Staubli VAL3: USERPAGE.pjx

--- USERPAGE.pjx ---
Parameters version=s7.6 stackSize=5000 millimeterUnit=true
Program file=changeValue.pgx
Program file=clear.pgx
Program file=divideString.pgx
Program file=editNumField.pgx
Program file=example.pgx
Program file=findPos.pgx
Program file=getListPosition.pgx
Program file=getMenu.pgx
Program file=getView.pgx
Program file=insertDialog.pgx
Program file=isListEmpty.pgx
Program file=leftPos.pgx
Program file=listadd.pgx
Program file=listcreate.pgx
Program file=listcursor.pgx
Program file=listdel.pgx
Program file=listempty.pgx
Program file=listevent.pgx
Program file=listframe.pgx
Program file=listins.pgx
Program file=listredraw.pgx
Program file=listupdate.pgx
Program file=midPos.pgx
Program file=nullKey.pgx
Program file=numCopy.pgx
Program file=printScroll.pgx
Program file=questionDialog.pgx
Program file=read.pgx
Program file=rightPos.pgx
Program file=scroll.pgx
Program file=selectNewField.pgx
Program file=setCenter.pgx
Program file=setMenu.pgx
Program file=setSizeList.pgx
Program file=setView.pgx
Program file=showBoolStatus.pgx
Program file=strfill.pgx
Program file=strfillchr.pgx
Program file=stringCopy.pgx
Program file=stringToArray.pgx
Program file=strlength.pgx
Program file=timerDialog.pgx
Program file=type.pgx
Program file=typeCenter.pgx
Program file=typeLen.pgx
Program file=typeMenu.pgx
Program file=yes_no.pgx
Program file=yes_no_cancel.pgx
Data file=userPage.dtx

--- USERPAGE.dtx ---
bool Show
bool bReadWrite[9]
  [0] = true
  [1] = true
  [2] = true
  [3] = true
  [4] = true
  [5] = true
  [6] = true
  [7] = true
  [8] = true
public bool bShowDialog
public bool bUseEscape
public bool bUseRefresh
public num nBottomX[2]
  [0] = 38
  [1] = 38
public num nBottomY = 12
num nFirst
num nKey = 270
num nOffSet
num nOldValue[2]
  [0] = 200
  [1] = 200
public num nPage = 100000
public num nParaAdjustType
num nTest
public num nToSuperV = -1
public num nTopX[2]
public num nTopY
public num nView
public string sItems[9]
  [0] = "使用真空压力传感器    > true "
  [1] = "传送带调速            > false"
  [2] = "距离上限距离1         > -110 mm"
  [3] = "距离上限距离2         > 20 mm"
  [4] = "Bypass个数            > 0"
  [5] = "Bypass前距离上限的距离> -200 mm"
  [6] = "沿传送带X方向偏移     > 0 mm"
  [7] = "沿传送带Y方向偏移     > 0 mm"
  [8] = "沿传送带Z方向偏移     > 0 mm"
string sMessage
public string sTitle = "出料传送带设置"
public string sToSuperV
string stest[11]
  [0] = "sbx"
  [1] = "sdfgsd"
  [2] = "bsfghsfh"
  [3] = "sdfgsdfg"
  [4] = "shsgh"
  [5] = "ghdfh"
  [6] = "snsfg"
  [7] = "sfgsg"
  [8] = "sfgsdfg"
  [9] = "sfgs"
  [10] = "dfsgs"
string stest2
string stest3

--- divideString.pgx ---
public program divideString(string& x_sMsg[] (dimensions=1), num& x_nLine[] (dimensions=1))
  local string l_sCopyMsg
  local num l_nLength
  local string l_sSwap
  local num l_nFlag
  local num l_nTotalFlag
  local string l_sCR
  local num l_nPosCR
  local num i
begin
  //
  //  using:
  // x_sMessage->  the message you want print to video
  // x_nLine->     the number of the line that will be use
  //
  //
  // CARRIAGE RETURN
  l_sCR="#"
  x_nLine=0
  //length of a line for a message
  l_nLength=38
  // copy the msg
  l_sCopyMsg=x_sMsg
  // first case
  call findPos(l_sCopyMsg,l_sCR,l_nPosCR)
  if (getDisplayLen(l_sCopyMsg)>l_nLength-1) or (l_nPosCR!=-1)
    // compose the message
    do
      l_sSwap=l_sCopyMsg
      // set the x_sMsg
      if size(x_sMsg)-1<x_nLine
        append(x_sMsg)
      endIf
      call findPos(l_sCopyMsg,l_sCR,l_nPosCR)
      //
      if (getDisplayLen(l_sCopyMsg)>l_nLength-1 or (l_nPosCR!=-1)) and x_nLine<8
        // divide the string
        l_nTotalFlag=0
        call findPos(l_sCopyMsg,l_sCR,l_nPosCR)
        //
        // divide the string
        //
        if l_nPosCR!=-1 and l_nPosCR<l_nLength
          // CARRIAGE RETURN
          call leftPos(l_sCopyMsg,l_nPosCR,l_sSwap)
          //l_sSwap=left(l_sCopyMsg,l_nPosCR)
          call rightPos(l_sCopyMsg,getDisplayLen(l_sCopyMsg)-(l_nPosCR)-1,l_sCopyMsg)
          //l_sCopyMsg=right(l_sCopyMsg,len(l_sCopyMsg)-(l_nPosCR)-1)
          if getDisplayLen(l_sSwap)==0
            l_sSwap=" "
          endIf
        else
          //
          // search for the space then return
          //
          do
            call findPos(l_sSwap," ",l_nFlag)
            //l_nFlag=find(l_sSwap," ")
            if l_nFlag!=-1 and l_nFlag<=l_nLength
              //l_sSwap=right(l_sSwap,len(l_sSwap)-l_nFlag-1)
              call rightPos(l_sSwap,getDisplayLen(l_sSwap)-l_nFlag-1,l_sSwap)
              l_nTotalFlag=l_nTotalFlag+l_nFlag+1
            else
              if l_nTotalFlag==0 and (l_nFlag==-1 or l_nFlag>l_nLength)
                l_nFlag=-1
                l_nTotalFlag=38
              endIf
            endIf
          until l_nTotalFlag>=l_nLength+2 or l_nFlag==-1
          // NORMAL
          if l_nTotalFlag==0
            // FULL LINE
            call leftPos(l_sCopyMsg,l_nLength,l_sSwap)
            //l_sSwap=left(l_sCopyMsg,l_nLength)
            //l_sCopyMsg=right(l_sCopyMsg,len(l_sCopyMsg)-l_nLength)
            call rightPos(l_sCopyMsg,getDisplayLen(l_sCopyMsg)-l_nLength,l_sCopyMsg)
          else
            // DIVIDE IT
            call leftPos(l_sCopyMsg,l_nTotalFlag-l_nFlag-2,l_sSwap)
            //l_sSwap=left(l_sCopyMsg,l_nTotalFlag-l_nFlag-2)
            //l_sCopyMsg=right(l_sCopyMsg,len(l_sCopyMsg)-(l_nTotalFlag-l_nFlag-1))
            call rightPos(l_sCopyMsg,getDisplayLen(l_sCopyMsg)-(l_nTotalFlag-l_nFlag-1),l_sCopyMsg)
          endIf
        endIf
        // set the string
        x_sMsg[x_nLine]=l_sSwap
        x_nLine=x_nLine+1
      else
        // limit the string
        call rightPos(l_sSwap,l_nLength,x_sMsg[x_nLine])
        //x_sMsg[x_nLine]=right(l_sSwap,l_nLength)
        l_sSwap=""
      endIf
    until l_sSwap==""
  endIf
end

--- editNumField.pgx ---
public program editNumField(string x_sTitle (dimensions=1), string& x_sItemName[] (dimensions=1), num& x_nItem[] (dimensions=1), num& x_nMin[] (dimensions=1), num& x_nMax[] (dimensions=1))
  local num j
  local num l_nSize
  local num l_nKey
  local string l_sEvent
  local num l_nIndex
  local num l_nField
  local string l_sItem
  local num i
  local string l_sEmpty[2]
  local string l_sString1
  local num l_nFollow
begin
  //  //clear & copy
  //  nView=nFirst=0
  //  call listempty()
  //  call numCopy(x_nItem,nOldValue)
  //  call numCopy(x_nItem,nOffSet)
  //  for j=0 to size(nOffSet)-1
  //    nOffSet[j]=0
  //  endFor
  //  // take the size
  //  l_nSize=size(x_sItemName)-1
  //  // create the LIST
  //  call setSizeList(2,max((6-l_nSize/2)-2,2)-2,20,min((l_nSize+1),12))
  //  call listcreate(x_sTitle)
  //  //
  //  // insert items
  //  //
  //  if nParaAdjustType==1
  //    for j=0 to l_nSize
  //      l_sItem=x_sItemName[j]
  //      if l_sItem!=""
  //        if j==9
  //          call strlength(l_sItem,10)
  //          if x_nItem[j]==0
  //            call listadd(l_sItem+": "+"关")
  //          else
  //            call listadd(l_sItem+": "+"开")
  //          endIf
  //        else
  //          call strlength(l_sItem,10)
  //          call listadd(l_sItem+": "+toString(".3",x_nItem[j]))
  //        endIf
  //        nOffSet[j]=nOffSet[max(j-1,0)]
  //      else
  //        nOffSet[j]=nOffSet[max(j-1,0)]+1
  //      endIf
  //    endFor
  //  endIf
  //  if nParaAdjustType==2
  //    for j=0 to l_nSize
  //      l_sItem=x_sItemName[j]
  //      if l_sItem!=""
  //        if j==7
  //          call strlength(l_sItem,10)
  //          if x_nItem[j]==0
  //            call listadd(l_sItem+": "+"关")
  //          else
  //            call listadd(l_sItem+": "+"开")
  //          endIf
  //        else
  //          call strlength(l_sItem,10)
  //          call listadd(l_sItem+": "+toString(".3",x_nItem[j]))
  //        endIf
  //        nOffSet[j]=nOffSet[max(j-1,0)]
  //      else
  //        nOffSet[j]=nOffSet[max(j-1,0)]+1
  //      endIf
  //    endFor
  //  endIf
  //  if nParaAdjustType==3
  //    for j=0 to l_nSize
  //      l_sItem=x_sItemName[j]
  //      if l_sItem!=""
  //        call strlength(l_sItem,10)
  //        call listadd(l_sItem+": "+toString(".3",x_nItem[j]))
  //        nOffSet[j]=nOffSet[max(j-1,0)]
  //      else
  //        nOffSet[j]=nOffSet[max(j-1,0)]+1
  //      endIf
  //    endFor
  //  endIf
  //  // update the list
  //  call listupdate(0)
  //  do
  //    call clear(0,13)
  //    call typeMenu(8,"OK")
  //    l_nKey=get()
  //    call listevent(l_nKey,l_nIndex,l_sEvent)
  //    // use the offset
  //    i=l_nIndex+nOffSet[max(l_nIndex,0)]
  //    // on Enter Key
  //    if nParaAdjustType==1
  //      if l_nKey==270
  //        if l_nIndex==9
  //          call listcursor(l_nIndex,false)
  //          if size(x_nMin)==size(x_nItem)
  //            // use min and max
  //            l_sEmpty[0]="关"
  //            l_sEmpty[1]="开"
  //            call changeValue(x_nItem[l_nIndex],x_nMin[l_nIndex],x_nMax[l_nIndex],15,nView+nTopY+1,l_sEmpty)
  //          else
  //            l_sEmpty[0]="关"
  //            l_sEmpty[1]="开"
  //            call changeValue(x_nItem[l_nIndex],x_nMin[l_nIndex],x_nMax[l_nIndex],15,nView+nTopY+1,l_sEmpty)
  //          endIf
  //          // UPDATE
  //          call listdel(l_nIndex)
  //          l_sItem=x_sItemName[l_nIndex]
  //          call strlength(l_sItem,10)
  //          call listins(l_sItem+": "+l_sEmpty[x_nItem[l_nIndex]],l_nIndex)
  //          call listupdate(l_nIndex-nView)
  //        else
  //          call listcursor(l_nIndex,false)
  //          if size(x_nMin)==size(x_nItem)
  //            // use min and max
  //            l_sEmpty[0]=""
  //            l_sEmpty[1]=""
  //            call changeValue(x_nItem[i],x_nMin[i],x_nMax[i],15,nView+nTopY+1,l_sEmpty)
  //          else
  //            call changeValue(x_nItem[i],x_nMin,x_nMax,15,nView+nTopY+1,l_sEmpty)
  //          endIf
  //          // UPDATE
  //          call listdel(l_nIndex)
  //          l_sItem=x_sItemName[i]
  //          call strlength(l_sItem,10)
  //          call listins(l_sItem+": "+toString(".3",x_nItem[i]),l_nIndex)
  //          call listupdate(l_nIndex-nView)
  //        endIf
  //      endIf
  //    endIf
  //    if nParaAdjustType==2
  //      if l_nKey==270
  //        if l_nIndex==7
  //          call listcursor(l_nIndex,false)
  //          if size(x_nMin)==size(x_nItem)
  //            // use min and max
  //            l_sEmpty[0]="关"
  //            l_sEmpty[1]="开"
  //            call changeValue(x_nItem[l_nIndex],x_nMin[l_nIndex],x_nMax[l_nIndex],15,nView+nTopY+1,l_sEmpty)
  //          else
  //            l_sEmpty[0]="关"
  //            l_sEmpty[1]="开"
  //            call changeValue(x_nItem[l_nIndex],x_nMin[l_nIndex],x_nMax[l_nIndex],15,nView+nTopY+1,l_sEmpty)
  //          endIf
  //          //UPDATE
  //          call listdel(l_nIndex)
  //          l_sItem=x_sItemName[l_nIndex]
  //          call strlength(l_sItem,10)
  //          call listins(l_sItem+": "+l_sEmpty[x_nItem[l_nIndex]],l_nIndex)
  //          call listupdate(l_nIndex-nView)
  //        else
  //          call listcursor(l_nIndex,false)
  //          if size(x_nMin)==size(x_nItem)
  //            // use min and max
  //            l_sEmpty[0]=""
  //            l_sEmpty[1]=""
  //            call changeValue(x_nItem[i],x_nMin[i],x_nMax[i],15,nView+nTopY+1,l_sEmpty)
  //          else
  //            call changeValue(x_nItem[i],x_nMin,x_nMax,15,nView+nTopY+1,l_sEmpty)
  //          endIf
  //          // UPDATE
  //          call listdel(l_nIndex)
  //          l_sItem=x_sItemName[i]
  //          call strlength(l_sItem,10)
  //          call listins(l_sItem+": "+toString(".3",x_nItem[i]),l_nIndex)
  //          call listupdate(l_nIndex-nView)
  //        endIf
  //      endIf
  //    endIf
  //    if nParaAdjustType==3
  //      if l_nKey==270
  //        //      if l_nIndex==7
  //        //        call listcursor(l_nIndex,false)
  //        //        if size(x_nMin)==size(x_nItem)
  //        //          // use min and max
  //        //          l_sEmpty[0]="关"
  //        //          l_sEmpty[1]="开"
  //        //          call changeValue(x_nItem[l_nIndex],x_nMin[l_nIndex],x_nMax[l_nIndex],15,nView+nTopY+1,l_sEmpty)
  //        //        else
  //        //          l_sEmpty[0]="关"
  //        //          l_sEmpty[1]="开"
  //        //          call changeValue(x_nItem[l_nIndex],x_nMin[l_nIndex],x_nMax[l_nIndex],15,nView+nTopY+1,l_sEmpty)
  //        //        endIf
  //        //        //UPDATE
  //        //        call listdel(l_nIndex)
  //        //        l_sItem=x_sItemName[l_nIndex]
  //        //        call strlength(l_sItem,10)
  //        //        call listins(l_sItem+": "+l_sEmpty[x_nItem[l_nIndex]],l_nIndex)
  //        //        call listupdate(l_nIndex-nView)
  //        //      else
  //        call listcursor(l_nIndex,false)
  //        if size(x_nMin)==size(x_nItem)
  //          // use min and max
  //          l_sEmpty[0]=""
  //          l_sEmpty[1]=""
  //          call changeValue(x_nItem[i],x_nMin[i],x_nMax[i],15,nView+nTopY+1,l_sEmpty)
  //        else
  //          call changeValue(x_nItem[i],x_nMin,x_nMax,15,nView+nTopY+1,l_sEmpty)
  //        endIf
  //        // UPDATE
  //        call listdel(l_nIndex)
  //        l_sItem=x_sItemName[i]
  //        call strlength(l_sItem,10)
  //        call listins(l_sItem+": "+toString(".3",x_nItem[i]),l_nIndex)
  //        call listupdate(l_nIndex-nView)
  //        //      endIf
  //      endIf
  //    endIf
  //    delay(0)
  //  until l_nKey==278 or l_nKey==255
  //  // escape use????
  //  if l_nKey==255
  //    bUseEscape=true
  //    call numCopy(nOldValue,x_nItem)
  //  else
  //    bUseEscape=false
  //  endIf
  //  // exit
  //  call nullKey(l_nKey)
end

--- example.pgx ---
program example()
  local num l_nKey
  local num l_nItem[2]
  local num l_nView[2]
  local string l_sItem
  local string l_sMsg
  local num i
  local bool l_bLarge
  local bool l_bQuit
  local string l_sMenu
  local num l_nSeconds
  local string l_sHourMinSec
  local num l_nItemExample[5]
  local num l_nMaxExample[5]
  local num l_nMinExample[5]
  local num l_nMenu
  local num l_nSelected[2]
  local bool l_bExit
  local num l_nFirst[2]
  local string l_sButton[2]
  local string l_sItemName[5]
begin
  //-----------------------------------------------------------------------
  //Header begin
  //Description of program
  //  This is an example for use this library.
  //  This example performs the following actions :
  //  - Run the fhmns program (converted of num seconds in string hour)
  //  - add, insert, delete, and select an Item with an updating of the menu.
  //  - change Menu (list of Items) with left and right keys
  //  - clear the menu
  //  - Run a simple list (no array) for just test the scrolling
  //
  //  The sequence is :
  //  - Creation of 2 string arrays for the lists of items
  //  - Start main loop
  //  -   Creation of the menu with 2 lists
  //  -   Reading events from the keyboard
  //  -     case TAB           : update the width of the list (enlarge/reduce)
  //  -     case left or right : update the item's list and change the menu
  //  -     case Enter         : displays the Item selected
  //  -     case F1 or ESC     : quit the program
  //  -     case F2            : clear th list
  //  -     case F3            : Run function wich converted seconds
  //                              -> string Hours:Min:Sec
  //  -     case F4            : test editNumField() function
  //  -     case F5            : creation of an other list : simple list
  //  -     case F6            : delete an Item
  //  -     case F7            : add an item at the end of the list
  //  -     case F8            : insert an item at the current position
  //  -   Update the Item's list
  //  -   Refresh the screen
  //
  //History
  //  Creation : 28-04-08 - f.Rob
  //Header end
  //-----------------------------------------------------------------------
  ////////////////  cls()
  ////////////////  userPage()
  ////////////////  //---------------------------------------------------
  ////////////////  // CREATION OF 2 STRING ARRAYS FOR THE LISTS OF ITEMS
  ////////////////  //---------------------------------------------------
  ////////////////  //Empty the two lists
  ////////////////  call stringCopy("",sExample1)
  ////////////////  call stringCopy("",sExample2)
  ////////////////  //Build the first list
  ////////////////  for i=0 to 19
  ////////////////    if sExample1!=""
  ////////////////      $dins(sExample1,size(sExample1))
  ////////////////    endIf
  ////////////////    sExample1[i]="Program "+toString("",i)
  ////////////////  endFor
  ////////////////  //Build the second list
  ////////////////  for i=0 to 14
  ////////////////    if sExample2!=""
  ////////////////      $dins(sExample2,size(sExample2))
  ////////////////    endIf
  ////////////////    sExample2[i]="Item "+toString("",i)
  ////////////////  endFor
  ////////////////  //----------------
  ////////////////  // START THE LOOP
  ////////////////  //----------------
  ////////////////  do
  ////////////////    //-------------------------------------
  ////////////////    // CREATION OF THE MENU WITH TWO LISTS
  ////////////////    //-------------------------------------
  ////////////////    title("userPage example")
  ////////////////    //Creation size of the list
  ////////////////    call setSizeList(20,0,18,11)
  ////////////////    //Enlarge/reduce the width of the list menu when tab is pressed
  ////////////////    call setView(l_bLarge)
  ////////////////    //Refresh the list
  ////////////////    call listCreate("Menu "+toString("",l_nMenu+1))
  ////////////////    switch l_nMenu
  ////////////////      //Insert all the array into the list
  ////////////////      case 0
  ////////////////        call listAdd(sExample1)
  ////////////////      break
  ////////////////      case 1
  ////////////////        call listAdd(sExample2)
  ////////////////      break
  ////////////////    endSwitch
  ////////////////    //Refresh cursor position - selected item
  ////////////////    call selectNewField(l_nSelected[l_nMenu],l_nItem[l_nMenu],l_nView[l_nMenu])
  ////////////////    //Menu
  ////////////////    l_sMenu="Exit,Clean,Conversion,Parameter,Simple list,Delete,Add,Insert"
  ////////////////    call stringToArray(l_sMenu,sMenu)
  ////////////////    if !l_bLarge
  ////////////////      //Set the menu at the Y position : 3
  ////////////////      call setMenu(sMenu,true,3)
  ////////////////    else
  ////////////////      //Displays the menu on the bottom side not on the left side
  ////////////////      call setMenu(sMenu,true,-1)
  ////////////////    endIf
  ////////////////    //-----------------------------------
  ////////////////    //  READING EVENTS FROM THE KEYBOARD
  ////////////////    //-----------------------------------
  ////////////////    l_nKey=get()
  ////////////////    call listEvent(l_nKey,l_nItem[l_nMenu],l_sItem)
  ////////////////    //Update the cursor position viewing on the screen
  ////////////////    //The two lists are independent so utilisation of an array with two elements
  ////////////////    l_nView[l_nMenu]=nView
  ////////////////    //Update the selection of the Item
  ////////////////    l_nSelected[l_nMenu]=l_nItem[l_nMenu]
  ////////////////    switch (l_nKey)
  ////////////////      //Tab
  ////////////////      //------------------------------------------------
  ////////////////      //  UPDATE THE WIDTH OF THE LIST (ENLARGE/REDUCE)
  ////////////////      //------------------------------------------------
  ////////////////      case 259
  ////////////////        //Variable corresponding to Enlarge/Reduce the width of the list
  ////////////////        l_bLarge=!l_bLarge
  ////////////////      break
  ////////////////      //Left or Right
  ////////////////      //---------------------------------------------
  ////////////////      //  UPDATE THE ITEM'S LIST AND CHANGE THE MENU
  ////////////////      //---------------------------------------------
  ////////////////      case 264,268
  ////////////////        switch l_nMenu
  ////////////////          case 0
  ////////////////            call stringCopy(sItems,sExample1)
  ////////////////          break
  ////////////////          case 1
  ////////////////            call stringCopy(sItems,sExample2)
  ////////////////          break
  ////////////////        endSwitch
  ////////////////        //Update l_nMenu
  ////////////////        if l_nKey==264
  ////////////////          //Right
  ////////////////          //Increment l_nMenu
  ////////////////          l_nMenu=abs(l_nMenu-1)%2
  ////////////////        else
  ////////////////          //Left
  ////////////////          //Decrement l_nMenu
  ////////////////          l_nMenu=abs(l_nMenu+1)%2
  ////////////////        endIf
  ////////////////        //Update the selected item
  ////////////////        l_nSelected[l_nMenu]=l_nItem[l_nMenu]
  ////////////////      break
  ////////////////      //Enter
  ////////////////      //-----------------------------
  ////////////////      //  DISPLAYS THE ITEM SELECTED
  ////////////////      //-----------------------------
  ////////////////      case 270
  ////////////////        //No action just displays a message, it's an example
  ////////////////        call timerDialog("Selected item: "+l_sItem,1)
  ////////////////      break
  ////////////////      //F1
  ////////////////      //-------------------
  //  QUIT THE PROGRAM
  //-------------------
  ////////////////      case 271
  ////////////////        //Creation of two buttons functions
  ////////////////        //l_sButton    : F8
  ////////////////        //l_sButton[1] : F7
  ////////////////        l_sButton="Yes"
  ////////////////        l_sButton[1]="No"
  ////////////////        call questionDialog("Do you want to quit ?",l_sButton,l_nKey)
  ////////////////        //"Enter" or "F8" pressed
  ////////////////        if l_nKey==0 or l_nKey==1
  ////////////////          l_bQuit=true
  ////////////////        endIf
  ////////////////        cls()
  ////////////////      break
  //F2
  //-----------------
  //  CLEAR THE LIST
  //-----------------
  //////////////////      case 272
  //////////////////        //Creation of two buttons functions
  //////////////////        //l_sButton    : F8
  //////////////////        //l_sButton[1] : F7
  //////////////////        l_sButton="Yes"
  //////////////////        l_sButton[1]="No"
  //////////////////        call questionDialog("Do you want to clear the list ?",l_sButton,i)
  //////////////////        if i==0 or i==1
  //////////////////          call listEmpty()
  //////////////////        endIf
  //////////////////      break
  //F3
  //--------------------------------------------------------------
  //  RUN FUNCTION WICH CONVERTED SECONDS -> STRING HOURS:MIN:SEC
  //--------------------------------------------------------------
  ////////////////      case 273
  ////////////////        cls()
  ////////////////        call insertDialog("Number of seconds that you want to convert in Hour:min:sec : #",l_nSeconds,0,0)
  ////////////////        call fhmns(l_nSeconds,l_sHourMinSec)
  ////////////////        popUpMsg("Conversion : "+l_sHourMinSec)
  ////////////////      break
  //F4
  //---------------------------------
  //  TEST " EDITNUMFIELD " FUNCTION
  //---------------------------------
  ////////////////      case 274
  ////////////////        //Test editNumField function
  ////////////////        for i=0 to size(l_sItemName)-1
  ////////////////          l_sItemName[i]="Item "+toString("",i)
  ////////////////          //No Limits for all
  ////////////////          l_nMinExample[i]=0
  ////////////////          l_nMaxExample[i]=0
  ////////////////        endFor
  ////////////////        call editNumField("Change Parameter",l_sItemName,l_nItemExample,l_nMinExample,l_nMaxExample)
  ////////////////      break
  // F5
  //------------------------------------------
  //  CREATION OF AN OTHER LIST : SIMPLE LIST
  //------------------------------------------
  ////////////////      case 275
  ////////////////        //Simple list for test the scrolling
  ////////////////        cls()
  ////////////////        do
  ////////////////          l_bExit=false
  ////////////////          //Size of the list
  ////////////////          call setSizeList(20,0,18,11)
  ////////////////          //Creation of the list with the title "Simple list"
  ////////////////          call listCreate("Simple list")
  ////////////////          //Add Items in the list
  ////////////////          call listAdd("Item 1")
  ////////////////          call listAdd("Item 2")
  ////////////////          call listAdd("Item 3")
  ////////////////          call listAdd("Item 4")
  ////////////////          //Update the list
  ////////////////          call listUpdate(0)
  ////////////////          call typeMenu(1,"Quit simple list")
  ////////////////          i=get()
  ////////////////          call listEvent(i,0,"")
  ////////////////          switch i
  ////////////////            case 271,255
  ////////////////              l_sButton="Yes"
  ////////////////              l_sButton[1]="No"
  ////////////////              call questionDialog("Do you want to quit this program ?",l_sButton,i)
  ////////////////              //"Enter" or "F8" pressed
  ////////////////              if i==0 or i==1
  ////////////////                l_bExit=true
  ////////////////              else
  ////////////////                cls()
  ////////////////              endIf
  ////////////////            break
  ////////////////          endSwitch
  ////////////////        until l_bExit
  ////////////////      break
  //F6
  //-----------------
  //  DELETE AN ITEM
  //-----------------
  ////////////////      case 276
  ////////////////        //Delete
  ////////////////        l_sButton="Yes"
  ////////////////        l_sButton[1]="No"
  ////////////////        call questionDialog("Do you want to delete "+l_sItem+" ?",l_sButton,i)
  ////////////////        if i==0 or i==1
  ////////////////          call listDel(l_nItem[l_nMenu])
  ////////////////        endIf
  ////////////////      break
  //F7
  //---------------------------------
  //  ADD AN ITEM AT END OF THE LIST
  //---------------------------------
  ////////////////      case 277
  ////////////////        call timerDialog("Add One element #",0)
  ////////////////        l_sItem="new Item"
  ////////////////        //Read one string from the keyboard and write it on the
  ////////////////        //15 column and 7 line.
  ////////////////        call read(15,7,l_sItem,10,false)
  ////////////////        if !bUseEscape
  ////////////////          call listAdd(l_sItem)
  ////////////////        endIf
  ////////////////        switch l_nMenu
  ////////////////          case 0
  ////////////////            l_nSelected=size(sExample1)
  ////////////////          break
  ////////////////          case 1
  ////////////////            l_nSelected=size(sExample2)
  ////////////////          break
  ////////////////        endSwitch
  ////////////////      break
  //F8
  //-----------------------------------------
  //  INSERT AN ITEM AT THE CURRENT POSITION
  //-----------------------------------------
  //////////////      case 278
  //////////////        //Insert at the current position
  //////////////        call timerDialog("Insert One element #",0)
  //////////////        l_sItem="new Item"
  //////////////        call read(15,7,l_sItem,10,false)
  //////////////        if !isKeyPressed(255) and l_sItem!="new Item"
  //////////////          call listIns(l_sItem,l_nItem[l_nMenu])
  //////////////        endIf
  //////////////      break
  //////////////    endSwitch
  //-------------------------
  //  UPDATE THE ITEM'S LIST
  //-------------------------
  //Update the list
  ////////////    switch l_nKey
  ////////////      case 272,276,277,278
  ////////////        //Update the item's list with the cycleStatus variable
  ////////////        switch l_nMenu
  ////////////          case 0
  ////////////            call stringCopy(sItems,sExample1)
  ////////////          break
  ////////////          case 1
  ////////////            call stringCopy(sItems,sExample2)
  ////////////          break
  ////////////        endSwitch
  ////////////      break
  ////////////    endSwitch
  //-------------------
  //REFRESH THE SCREEN
  //-------------------
  ////////////    if l_nKey>=270 and l_nKey<=278 or l_nKey==259
  ////////////      cls()
  ////////////    endIf
  ////////////    delay(0)
  ////////////  until l_bQuit
end

--- insertDialog.pgx ---
public program insertDialog(string x_sMsg (dimensions=1), num& x_nItem[] (dimensions=1), num x_nMin (dimensions=1), num x_nMax (dimensions=1))
  local num l_nStartLine
  local num l_nLine
  local num i
  local num l_nPX
  local num l_nPY
  local string l_sItem
  local string l_sMessage
  local string l_sEmpty
  local string l_sCopy
begin
  //
  // modify the x_sItem, using a min max range
  //
  if watch(bShowDialog==false,2)==false
    bShowDialog=false
    logMsg("error dialog resoursing")
    return
  else
    setMutex(bShowDialog)
    // clear the line
    call clear(0,13)
    // look for the comma
    if round(x_nItem)!=x_nItem
      l_sItem=toString(".2",x_nItem)
    else
      l_sItem=toString("",x_nItem)
    endIf
    // print the line
    l_sCopy=x_sMsg+">"+l_sItem
    call stringCopy(l_sCopy,sMessage)
    // divide the sentence
    call divideString(sMessage,l_nLine)
    l_nStartLine=round(5-l_nLine/2)
    // Start LINE
    call type(0,l_nStartLine-2,"┌──────────────────────────────────────┐")
    call type(0,l_nStartLine-1,"│                                      │")
    // write the message
    for i=0 to l_nLine
      //call type(,"                                      ")
      l_sMessage=sMessage[i]
      call typeCenter(i+l_nStartLine,l_sMessage,38,false)
      call type(0,l_nStartLine+i,"│"+l_sMessage+"│")
    endFor
    // end LINE
    call type(0,l_nStartLine+l_nLine+1,"│                                      │")
    call type(0,l_nStartLine+l_nLine+2,"└──────────────────────────────────────┘")
    l_nPX=find(l_sMessage,">")+2
    l_nPY=l_nStartLine+l_nLine
    // change the value
    call changeValue(x_nItem,x_nMin,x_nMax,l_nPX,l_nPY,l_sEmpty)
    //
    bShowDialog=false
    bUseRefresh=true
    //
    delay(0)
  endIf
end

--- listcursor.pgx ---
public program listcursor(num pView (dimensions=1), bool pShow (dimensions=1))
  local num lX
  local num lY
  local string message
  local bool l_bEmpty
begin
  //
  // toneage Staubli Copyright 2005
  //
  call isListEmpty(l_bEmpty)
  if !l_bEmpty
    nView=pView
    lX=nTopX+1
    lY=nTopY+1+pView
    if (nView+nFirst)>(size(sItems)-1)
      call strfill(sItems[size(sItems)-1],nBottomX,message)
    else
      call strfill(sItems[nView+nFirst],nBottomX,message)
    endIf
    gotoxy(lX,lY)
    if (pShow==true)
      setTextMode(1)
      put(message)
      setTextMode(0)
    else
      setTextMode(0)
      put(message)
    endIf
  endIf
end

--- listempty.pgx ---
public program listempty()
  local num lI
  local num lLen
  local string lRun[5]
  local num lRuni
begin
  //
  // Staubli Copyright 2003 06 20
  //
  lLen=size(sItems)-1
  for lI=0 to lLen
    if lI>0
      $ddel(sItems,0)
      $ddel(bReadWrite,0)
    endIf
  endFor
  sItems=""
  //
end

--- listevent.pgx ---
public program listevent(num pkey (dimensions=1), num& pIndex[] (dimensions=1), string& pItem[] (dimensions=1))
  local num lVal
  local num l_nSize
  local bool l_bEmpty
begin
  //
  // Toneage Staubli product
  //
  //
  // get the item in the list and scroll it
  //
  call isListEmpty(l_bEmpty)
  if !l_bEmpty
    l_nSize=size(sItems)-1
    // check the overFlow
    l_nSize=size(sItems)-1
    if (nFirst+nView>l_nSize)
      // reset the value
      nFirst=nView=0
    endIf
    // security...
    switch (pkey)
      //Up
      case 261
        if ((nView-1)>=0)
          // no need to scroll only change cursor position
          call listcursor(nView,false)
          nView=nView-1
          call listcursor(nView,true)
          // print the scroll
          //call printScroll()
        else
          if nView==0
            // scroll up
            if ((nFirst-1)>=0)
              nFirst=nFirst-1
              call listupdate(nFirst)
            else
              // go to the end
              if nView+nFirst!=l_nSize
                call listcursor(nView,false)
                call selectNewField(l_nSize,nFirst+nView,nView)
              endIf
            endIf
          endIf
        endIf
      break
      //Down
      case 266
        if ((nView+nFirst+1)<size(sItems))
          // no need to scroll only chenge cursor position
          if ((nView+1)<nBottomY)
            call listcursor(nView,false)
            nView=nView+1
            call listcursor(nView,true)
            // print the scroll
            //call printScroll()
          else
            // move UP
            nFirst=nFirst+1
            call listupdate(nFirst)
          endIf
        else
          // go to the top
          if !(nView==0 and nFirst==0)
            call listcursor(nView,false)
            nView=0
            call listupdate(0)
          endIf
        endIf
      break
      //Page Up
      case 262
        if !(nView==0 and nFirst==0)
          call listcursor(nView,false)
          if ((nFirst+nView-nBottomY)>=0)
            // move one page up
            call selectNewField(nFirst+nView-nBottomY,nFirst+nView,nView)
          else
            // go to home
            nView=0
            call listupdate(0)
          endIf
        endIf
      break
      //Page Down
      case 267
        if nView+nFirst!=l_nSize
          call listcursor(nView,false)
          if ((nView+nFirst+nBottomY)<size(sItems)-1)
            // move one page down
            call selectNewField(nFirst+nView+nBottomY,nFirst+nView,nView)
          else
            // go to the end
            call selectNewField(l_nSize,nFirst+nView,nView)
          endIf
        endIf
      break
      //End
      case 269
        if nView+nFirst!=l_nSize
          // move to end
          call listcursor(nView,false)
          call selectNewField(l_nSize,nFirst+nView,nView)
        endIf
      break
      //Home
      case 265
        if !(nView==0 and nFirst==0)
          // move to home
          call listcursor(nView,false)
          nView=0
          call listupdate(0)
        endIf
      break
      default
      break
    endSwitch
    pIndex=nFirst+nView
    pItem=sItems[pIndex]
    //
  else
    // reset the item
    pItem=""
    pIndex=0
  endIf
end

--- listframe.pgx ---
program listframe(string pTitle (dimensions=1), num pX (dimensions=1), num pY (dimensions=1), num pDx (dimensions=1), num pDy (dimensions=1))
  local num lDx
  local num lDy
  local num lI
  local num lJ
  local string lStr
  local string lStrLine
  local num lValue
begin
  //
  // Staubli Copyright 2003 06 20
  //
  lStrLine="─────────────────────────────────────────"
  lDx=pDx
  lDy=pDy
  //Top
  lStr="┌"+mid(lStrLine,lDx,0)+"┐"
  gotoxy(pX,pY)
  put(lStr)
  lValue=pX+2
  //Title
  if pTitle!=""
    call leftPos("┤"+pTitle+"├",lDx,pTitle)
    gotoxy(pX+lDx-getDisplayLen(pTitle)+1,pY)
    put(pTitle)
  endIf
  //Containt
  for lJ=1 to lDy
    lValue=pY+lJ
    lStr="│"
    gotoxy(pX,lValue)
    put(lStr)
    gotoxy(pX+lDx+1,lValue)
    put(lStr)
  endFor
  //Bottom
  lValue=pY+lJ
  lStr="└"+mid(lStrLine,lDx,0)+"┘"
  gotoxy(pX,lValue)
  put(lStr)
end

--- listupdate.pgx ---
public program listupdate(num pFirst)
  local num lI
  local num lLen
  local string lStr
  local string lStr2
  local num lValue
  local num lView
  local num lX
  local num lY
  local num l_nSize
  local bool l_bEmpty
begin
  //
  // insert into the box all the data
  //
  // to prevent a negative value
  if pFirst>=0
    nFirst=pFirst
  else
    nFirst=0
  endIf
  // save the coordinate
  lValue=nBottomY-1
  // check the overFlow
  l_nSize=size(sItems)-1
  if (nFirst+nView>l_nSize)
    // reset the value
    nFirst=nView=0
  endIf
  lI=0
  // check the unKnow poblem
  if l_nSize<lValue
    if nFirst!=0
      nView=nView+nFirst
      nFirst=0
    endIf
  endIf
  do
    lX=nTopX+1
    lY=nBottomY+lI-1
    lY=nTopY+lI+1
    lLen=nBottomX
    if ((lI+nFirst)<size(sItems))
      // print the item
      if (l_nSize>=0)
        lStr=mid(sItems[(lI+nFirst)],lLen,0)
      endIf
    else
      // print the blank line
      lStr="                                        "
    endIf
    // fill the line
    call strfill(lStr,lLen,lStr2)
    gotoxy(lX,lY)
    put(lStr2)
    lI=lI+1
  until (lI>lValue)
  // underlien the actual line
  call isListEmpty(l_bEmpty)
  if !l_bEmpty
    call listcursor(nView,true)
  else
    call listcursor(nView,false)
    nView=0
    nFirst=0
  endIf
  // print the scroll
  call printScroll()
  // leave the resourse
  delay(0)
end

--- printScroll.pgx ---
program printScroll()
  local num i
  local num lX
  local num lY
begin
  //
  // put the scroll
  //
  if size(sItems)>nBottomY
    // find the percentage
    //windows style
    //i=(size(sItems)-nBottomY+1)/(nFirst+1)
    // nokia style
    i=(size(sItems))/(nFirst+nView+1)
    lX=nTopX+nBottomX+1
    lY=roundUp((nBottomY)/i+nTopY)
    for i=nTopY+1 to nBottomY
      gotoxy(lX,i)
      if i==lY
        //
        put("■")
      else
        put("│")
      endIf
    endFor
  endIf
end

--- questionDialog.pgx ---
public program questionDialog(string x_sMsg (dimensions=1), string& x_sButton[] (dimensions=1), num& x_nResult[] (dimensions=1))
  local bool lExit
  local num nLine
  local num i
  local num nStartLine
  local string l_sMessage
begin
  //---------------------------------
  //      D I A L O G    B O X
  //---------------------------------
  //
  // Show one dialog box. with an confirm question
  //
  if watch(bShowDialog==false,2)==false
    bShowDialog=false
    logMsg("error dialog resoursing")
    return
  else
    setMutex(bShowDialog)
    //call listempty()
    //
    //
    if x_sMsg!=""
      call stringCopy(x_sMsg,sMessage)
      call divideString(sMessage,nLine)
      nStartLine=round(5-nLine/2)
      // Start LINE
      call type(0,nStartLine-2,"┌──────────────────────────────────────┐")
      call type(0,nStartLine-1,"│                                      │")
      // write the message
      for i=0 to nLine
        l_sMessage=sMessage[i]
        call typeCenter(i+nStartLine,l_sMessage,38,false)
        call type(0,nStartLine+i,"│"+l_sMessage+"│")
      endFor
      // end LINE
      call type(0,nStartLine+nLine+1,"│                                      │")
      call type(0,nStartLine+nLine+2,"└──────────────────────────────────────┘")
    endIf
    // write the button message
    call clear(0,13)
    for i=0 to size(x_sButton)-1
      call typeMenu(8-i,x_sButton[i])
    endFor
    lExit=false
    x_nResult=-100
    do
      nKey=get()
      switch (nKey)
        case 270
          x_nResult=0
        break
        case 255
          x_nResult=-1
          bUseEscape=true
        break
        default
          // look if the button press is defined
          if (nKey>=271 and nKey<=278) and ((279-nKey)<=size(x_sButton))
            if x_sButton[278-nKey]!=""
              x_nResult=279-nKey
            endIf
          endIf
        break
      endSwitch
      delay(0)
    until (x_nResult!=-100)
    //
    call nullKey(nKey)
    //
    // release
    bShowDialog=false
    bUseRefresh=true
  endIf
end
